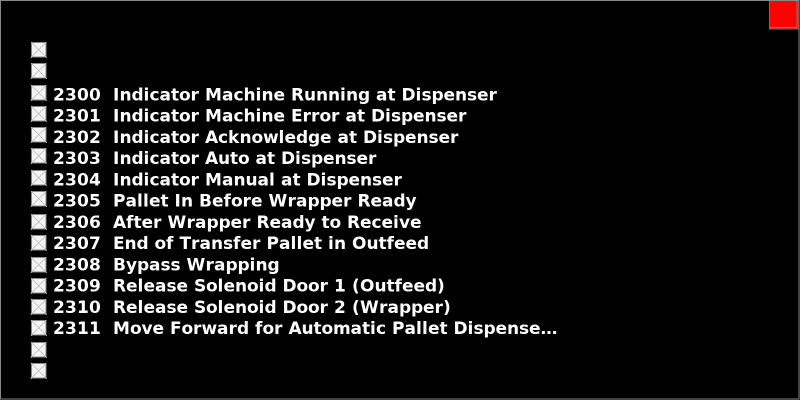
VISUALIZATION P2_DO4  // 800x400, background image 
    ImageSwitcher (31,42 15x15), variable: InputOutput_GVL.Digital_Output[49], behaviour: TOGGLE
    Label (50,16 625x391), "2300 Indicator Machine Running at Dispenser 2301 Indicator Machine Error at Dispenser 2302 Indicator Acknowledge at Dispenser 2303 Indicator Auto at Dispenser 2304 Indicator Manual at Dispenser 2305 Pallet In Before Wrapper Ready 2306 After Wrapper Ready to Receive 2307 End of Transfer Pallet in Outfeed 2308 Bypass Wrapping 2309 Release Solenoid Door 1 (Outfeed) 2310 Release Solenoid Door 2 (Wrapper) 2311 Move Forward for Automatic Pallet Dispenser 2312 Pneumatic Vertical Up 2313 Pneumatic Vertical Down 2314 Pneumatic Horizontal Rectract 2315 Pneumatic Horizontal Advanced"
    ImageSwitcher (31,63 15x15), variable: InputOutput_GVL.Digital_Output[50], behaviour: TOGGLE
    ImageSwitcher (31,85 15x15), variable: InputOutput_GVL.Digital_Output[51], behaviour: TOGGLE
    ImageSwitcher (31,106 15x15), variable: InputOutput_GVL.Digital_Output[52], behaviour: TOGGLE
    ImageSwitcher (31,127 15x15), variable: InputOutput_GVL.Digital_Output[53], behaviour: TOGGLE
    ImageSwitcher (31,148 15x15), variable: InputOutput_GVL.Digital_Output[54], behaviour: TOGGLE
    ImageSwitcher (31,170 15x15), variable: InputOutput_GVL.Digital_Output[55], behaviour: TOGGLE
    ImageSwitcher (31,191 15x15), variable: InputOutput_GVL.Digital_Output[56], behaviour: TOGGLE
    ImageSwitcher (31,214 15x15), variable: InputOutput_GVL.Digital_Output[57], behaviour: TOGGLE
    ImageSwitcher (31,235 15x15), variable: InputOutput_GVL.Digital_Output[58], behaviour: TOGGLE
    ImageSwitcher (31,257 15x15), variable: InputOutput_GVL.Digital_Output[59], behaviour: TOGGLE
    ImageSwitcher (31,278 15x15), variable: InputOutput_GVL.Digital_Output[60], behaviour: TOGGLE
    ImageSwitcher (31,299 15x15), variable: InputOutput_GVL.Digital_Output[61], behaviour: TOGGLE
    ImageSwitcher (31,320 15x15), variable: InputOutput_GVL.Digital_Output[62], behaviour: TOGGLE
    ImageSwitcher (31,342 15x15), variable: InputOutput_GVL.Digital_Output[63], behaviour: TOGGLE
    ImageSwitcher (31,363 15x15), variable: InputOutput_GVL.Digital_Output[64], behaviour: TOGGLE
    Button (769,-1 30x30), image: VisuSymbols.Symbols.Wrong
        OnMouseClick: CloseDialog Dialog=P2_DO4, Result=OK, NumpadKeypadSet=True
END_VISUALIZATION

(* stored: Version 1.1.0.1, ProductVersion 3.1.4024.12
   Visu P2_DO4: Id {22a76660-7056-4b83-b06a-04949e5cd5e6} *)
